(* CoDeSys 2.3.9.59 project: TwinatAds.pro *)
(* Libraries: STANDARD.LIB 5.6.98 11:03:02 *)

(* Task configuration *)
TASK Standard (PRIORITY := 0, INTERVAL := T#4ms);
	MAIN
END_TASK

(* Global variable list: Global_Variables *)
VAR_GLOBAL
	(* variable test  *)
	junit_bit					:BOOL;
	junit_int8					:SINT;
	junit_int16				:INT;
	junit_int32				:DINT;
	junit_uint8				:BYTE;
	junit_uint16				:WORD;
	junit_uint32				:DWORD;
	junit_real32				:REAL;
	junit_real64				:LREAL;
	junit_string				:STRING(100);

	(* loader test  *)
	junit_array_simple			:ARRAY[0..2, 2..4, 4..6] OF INT;
	junit_array_complex		:ARRAY[0..2, 4..8] OF fb_junit;
	junit_function_block		:fb_junit;
	juint_struct				:junit_st;

	(* problem *)
	junit_time					:TIME;
	juinit_p_simple			:POINTER TO LREAL;
	juinit_p_complex			:POINTER TO junit_st;
	juinit_p_complex_array 	:POINTER TO ARRAY [0..2] OF junit_st;
END_VAR

VAR_GLOBAL CONSTANT
	junit_c			:INT := 10;
END_VAR

(* Data type *)
TYPE junit_st :
STRUCT
	b_value		:BOOL;
	st_value		:TON;
END_STRUCT
END_TYPE

(* POU main, ST *)
PROGRAM main
VAR
END_VAR
;
END_PROGRAM

(* POU fb_junit, ST *)
FUNCTION_BLOCK fb_junit
VAR_INPUT
	input	:BOOL;
END_VAR

VAR_OUTPUT
	output	:LREAL;
END_VAR

VAR
	internal_structure			:junit_st;
	internal_primitive			:INT;
	internal_primitive_array		:ARRAY [0..2] OF BOOL;
	internal_structure_array		:ARRAY [1..3] OF junit_st;
END_VAR
;
END_FUNCTION_BLOCK
